{attribute 'qualified_only'}
VAR_GLOBAL CONSTANT
	BUFFER_SIZE : INT := (100 * UDINT_TO_INT(MAX_STRING_LENGTH));
END_VAR

(* stored: Version 1.1.0.1
   GVL CONSTANTS: Id {98d3c9eb-cf89-468b-a8b6-e3b4bfd38910}, ParameterList True *)
